(* CODESYS project tom_2_8_RECOVERED_2024-06-01T16-58-33.project

Project tree, tasks and I/O mapping:
  Device : CODESYS Control Win V3, CODESYS, version 3.5.20.0
    application Application
      libraries: Standard, 3.5.18.0 (System)
      task MainTask (cyclic, interval t#20ms, priority 1) calls PLC_PRG
      program PLC_PRG [LD]
*)

// Device/Application/PLC_PRG
PROGRAM PLC_PRG
VAR
	S1: BOOL;
	P1: BOOL;
	S2: BOOL;
	P2: BOOL;
END_VAR

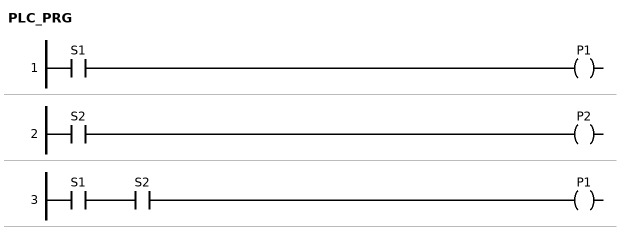
// NETWORK 1
P1 := S1;

// NETWORK 2
P2 := S2;

// NETWORK 3
P1 := S1 AND S2;

END_PROGRAM
